// TIA Portal V18 export
VAR_GLOBAL   // PLC tag table "Alarms"
   "Alarm Main 1/5" AT %MW600 : Word;
   "Alarm Main 2/5" AT %MW602 : Word;
   "Alarm Main 3/5" AT %MW604 : Word;
   "Alarm Main 4/5" AT %MW606 : Word;
   "Alarm Main 5/5" AT %MW608 : Word;
   "Alarm Main 6" AT %MW610 : Word;
   "Alarm Main 7" AT %MW612 : Word;
   "AL-AutoLeveller Down" AT %M614.0 : Bool;
   "AL-AutoLeveller Down Over Work" AT %M607.2 : Bool;
   "AL-AutoLeveller Motor Fault" AT %M607.7 : Bool;
   "AL-AutoLeveller Touch" AT %M607.3 : Bool;
   "AL-AutoLeveller Up" AT %M614.1 : Bool;
   "AL-AutoLeveller Up Over Work" AT %M607.1 : Bool;
   "AL-ByPass Activated" AT %M611.1 : Bool;
   "AL-Cab Floor BW Button Pressed" AT %M610.1 : Bool;
   "AL-Cab Floor FW Button Pressed" AT %M610.0 : Bool;
   "AL-Cab Floor Motor Fault" AT %M610.2 : Bool;
   "AL-Cab Left Button Pressed" AT %M609.6 : Bool;
   "AL-Cab Left Stop Limit, All" AT %M609.0 : Bool;
   "AL-Cab Left Stop Limit, Angle" AT %M608.7 : Bool;
   "AL-Cab Left Stop Limit, LS" AT %M608.6 : Bool;
   "AL-Cab Motor MKS" AT %M609.5 : Bool;
   "AL-Cab Right Button Pressed" AT %M609.7 : Bool;
   "AL-Cab Right Stop Limit, All" AT %M609.3 : Bool;
   "AL-Cab Right Stop Limit, Angle" AT %M609.2 : Bool;
   "AL-Cab Right Stop Limit, LS" AT %M609.1 : Bool;
   "AL-Canopy BW Button Pressed" AT %M608.5 : Bool;
   "AL-Canopy FW Button Pressed" AT %M608.4 : Bool;
   "AL-CP Emergency Stop Pressed" AT %M610.7 : Bool;
   "AL-Down Button Pressed" AT %M607.6 : Bool;
   "AL-Down Stop Limit, All" AT %M606.6 : Bool;
   "AL-Down Stop Limit, FW LS" AT %M606.5 : Bool;
   "AL-Down Stop Limit, Min Slope" AT %M606.4 : Bool;
   "AL-Down Stop Limit, Object" AT %M606.3 : Bool;
   "AL-Down Stop Limit, Wire" AT %M606.2 : Bool;
   "AL-Drive Angle LS BW Stop" AT %M619.4 : Bool;
   "AL-Drive Angle LS FW Stop" AT %M619.5 : Bool;
   "AL-Drive Left Slow Limit Angle" AT %M600.0 : Bool;
   "AL-Drive Left Stop Limit" AT %M600.3 : Bool;
   "AL-Drive Left Stop Limit Angle" AT %M600.2 : Bool;
   "AL-Drive Left Stop Limit LS" AT %M600.1 : Bool;
   "AL-Drive Right Slow Limit Angle" AT %M600.4 : Bool;
   "AL-Drive Right Stop Limit" AT %M600.7 : Bool;
   "AL-Drive Right Stop Limit Angle" AT %M600.6 : Bool;
   "AL-Drive Right Stop Limit LS" AT %M600.5 : Bool;
   "AL-Drive Slow Limit All" AT %M604.7 : Bool;
   "AL-Driver Fault, Cab" AT %M609.4 : Bool;
   "AL-Drivers Fault, Wheel" AT %M605.4 : Bool;
   "AL-Emergency Stop Pressed" AT %M611.0 : Bool;
   "AL-FAULT" AT %M611.4 : Bool;
   "AL-Hydraulic Motor MKS" AT %M607.4 : Bool;
   "AL-Left Canopy MKS" AT %M608.2 : Bool;
   "AL-Left Canopy Touch" AT %M608.0 : Bool;
   "AL-Left Emergency Stop Pressed" AT %M610.5 : Bool;
   "AL-Main Contactor ON" AT %M611.3 : Bool;
   "AL-No Electricity" AT %M611.6 : Bool;
   "AL-PBB HOME" AT %M619.6 : Bool;
   "AL-PBB in Auto Mode" AT %M610.4 : Bool;
   "AL-PBB in Off Mode" AT %M610.3 : Bool;
   "AL-PBB in On Mode" AT %M611.2 : Bool;
   "AL-Right Canopy MKS" AT %M608.3 : Bool;
   "AL-Right Canopy Touch" AT %M608.1 : Bool;
   "AL-Right Emergency Stop Pressed" AT %M610.6 : Bool;
   "AL-Rotunda BW Stop Limit All" AT %M602.2 : Bool;
   "AL-Rotunda FW Stop Limit All" AT %M602.1 : Bool;
   "AL-Rotunda Left BW Stop Limit" AT %M601.5 : Bool;
   "AL-Rotunda Left FW Stop Limit" AT %M601.4 : Bool;
   "AL-Rotunda Left Slow Limit" AT %M601.0 : Bool;
   "AL-Rotunda Left Stop Limit LS" AT %M601.3 : Bool;
   "AL-Rotunda Right BW Stop Limit" AT %M602.0 : Bool;
   "AL-Rotunda Right FW Stop Limit" AT %M601.7 : Bool;
   "AL-Rotunda Right Slow Limit" AT %M601.1 : Bool;
   "AL-Rotunda Right Stop Limit LS" AT %M601.6 : Bool;
   "AL-Rotunda Slow Limit" AT %M601.2 : Bool;
   "AL-SafetyBarrier Activated" AT %M611.5 : Bool;
   "AL-SafetyShoe Activated" AT %M606.7 : Bool;
   "AL-SafetyShoe Cable Problem" AT %M607.0 : Bool;
   "AL-Service" AT %M619.3 : Bool;
   "AL-Service-GPU" AT %M619.1 : Bool;
   "AL-Service-Hose" AT %M619.0 : Bool;
   "AL-Service-PCA" AT %M619.2 : Bool;
   "AL-Slow Activated" AT %M604.6 : Bool;
   "AL-Tunnel BW Emergency Stop Limit" AT %M604.5 : Bool;
   "AL-Tunnel BW Slow Limit All" AT %M603.2 : Bool;
   "AL-Tunnel BW Slow Limit Laser" AT %M603.0 : Bool;
   "AL-Tunnel BW Slow Limit LS" AT %M603.1 : Bool;
   "AL-Tunnel BW Slow Limit Slope" AT %M605.2 : Bool;
   "AL-Tunnel BW Stop Limit All" AT %M604.4 : Bool;
   "AL-Tunnel BW Stop Limit Laser" AT %M604.2 : Bool;
   "AL-Tunnel BW Stop Limit LS" AT %M604.3 : Bool;
   "AL-Tunnel BW Stop Limit Slope" AT %M605.3 : Bool;
   "AL-Tunnel FW Emergency Stop Limit" AT %M604.1 : Bool;
   "AL-Tunnel FW Slow Limit All" AT %M602.7 : Bool;
   "AL-Tunnel FW Slow Limit Laser" AT %M602.3 : Bool;
   "AL-Tunnel FW Slow Limit LS" AT %M602.4 : Bool;
   "AL-Tunnel FW Slow Limit PhotoCell" AT %M602.5 : Bool;
   "AL-Tunnel FW Slow Limit Slope" AT %M605.0 : Bool;
   "AL-Tunnel FW Slow Limit UltraSonic" AT %M602.6 : Bool;
   "AL-Tunnel FW Stop Limit All" AT %M604.0 : Bool;
   "AL-Tunnel FW Stop Limit Laser" AT %M603.3 : Bool;
   "AL-Tunnel FW Stop Limit LS" AT %M603.4 : Bool;
   "AL-Tunnel FW Stop Limit PhotoCell Left" AT %M603.5 : Bool;
   "AL-Tunnel FW Stop Limit PhotoCell Mid" AT %M603.6 : Bool;
   "AL-Tunnel FW Stop Limit PhotoCell Right" AT %M603.7 : Bool;
   "AL-Tunnel FW Stop Limit Slope" AT %M605.1 : Bool;
   "AL-Up Button Pressed" AT %M607.5 : Bool;
   "AL-Up Stop Limit, All" AT %M606.1 : Bool;
   "AL-Up Stop Limit, BW LS" AT %M606.0 : Bool;
   "AL-Up Stop Limit, Max Slope" AT %M605.7 : Bool;
   "AL-Up Stop Limit, Wire" AT %M605.6 : Bool;
   "AL-Wheel Fuse" AT %M605.5 : Bool;
   "AL-SafetyShoe Box Status" AT %M614.2 : Bool;
END_VAR
